FUNCTION_BLOCK "FB_Map_Siwarex_Core"
TITLE = Маппинг данных Siwarex CS
{ S7_Optimized_Access := 'FALSE' }
AUTHOR : S7C_Lib
FAMILY : Analog
VERSION : 1.4
// ==============================================================================
// Описание: Адаптированный маппинг из UDT_SIWA_CS. Обработка раздельных кодов
//           ошибок (модуля и драйвера). Встроенный таймер Watchdog в STAT.
// ==============================================================================
   VAR
      stat_Diag_CS_1 { ExternalAccessible := 'False'; ExternalVisible := 'False'; ExternalWritable := 'False'} : Struct   // Внутренняя память для Watchdog
         Old_Count { ExternalAccessible := 'False'; ExternalVisible := 'False'; ExternalWritable := 'False'} : Byte;
         Old_Weight { ExternalAccessible := 'False'; ExternalVisible := 'False'; ExternalWritable := 'False'} : Real;
         Last_Change_ms { ExternalAccessible := 'False'; ExternalVisible := 'False'; ExternalWritable := 'False'} : Real;
      END_STRUCT;
      stat_Diag_CS_2 { ExternalAccessible := 'False'; ExternalVisible := 'False'; ExternalWritable := 'False'} : Struct   // Внутренняя память для Watchdog
         Old_Count { ExternalAccessible := 'False'; ExternalVisible := 'False'; ExternalWritable := 'False'} : Byte;
         Old_Weight { ExternalAccessible := 'False'; ExternalVisible := 'False'; ExternalWritable := 'False'} : Real;
         Last_Change_ms { ExternalAccessible := 'False'; ExternalVisible := 'False'; ExternalWritable := 'False'} : Real;
      END_STRUCT;
   END_VAR

   VAR_TEMP
      temp_Value_Changed : Bool;
      temp_Counter_Changed : Bool;
   END_VAR


BEGIN

	// ============================================================================
	// SCALE CS_1
	// ============================================================================

	// 1. Веса
	"DB_MAP".Scale_CS_1.Weight_Gross_kg := INT_TO_REAL("DB_SCALE_CS_1".s_PROCESS_VALUES.i_GROSS_WEIGHT_PROC);
	"DB_MAP".Scale_CS_1.Weight_Net_kg := INT_TO_REAL("DB_SCALE_CS_1".s_PROCESS_VALUES.i_NET_WEIGHT_PROC);
	"DB_MAP".Scale_CS_1.Weight_Tare_kg := INT_TO_REAL("DB_SCALE_CS_1".s_PROCESS_VALUES.i_TARE_WEIGHT_PROC);

	// 2. Статусы
	"DB_MAP".Scale_CS_1.Status.Standstill := "DB_SCALE_CS_1".s_PROCESS_VALUES.bo_STA_ST_STAND_SCALE_ON;
	"DB_MAP".Scale_CS_1.Status.Limit_1 := "DB_SCALE_CS_1".s_PROCESS_VALUES.bo_STA_LIMIT1_ON;
	"DB_MAP".Scale_CS_1.Status.Limit_2 := "DB_SCALE_CS_1".s_PROCESS_VALUES.bo_STA_LIMIT2_ON;
	"DB_MAP".Scale_CS_1.Status.Tared := "DB_SCALE_CS_1".s_PROCESS_VALUES.bo_STA_TARED;
	"DB_MAP".Scale_CS_1.Status.Quarter_D_Zero := "DB_SCALE_CS_1".s_PROCESS_VALUES.bo_STA_025_D_ZERO;
	"DB_MAP".Scale_CS_1.Status.Scale_Calibrated := "DB_SCALE_CS_1".s_PROCESS_VALUES.bo_STA_SCALE_CALIBRATED;
	"DB_MAP".Scale_CS_1.Status.Write_Protected := "DB_SCALE_CS_1".s_PROCESS_VALUES.bo_STA_WRI_PROT;
	"DB_MAP".Scale_CS_1.Status.Limit_Max := "DB_SCALE_CS_1".s_PROCESS_VALUES.bo_STA_MAX_9E;
	"DB_MAP".Scale_CS_1.Status.Fault_HW := "DB_SCALE_CS_1".s_PROCESS_VALUES.bo_STA_ERROR_ON;
	"DB_MAP".Scale_CS_1.Status.Fault_FB := "DB_SCALE_CS_1".bo_FB_ERR;
	"DB_MAP".Scale_CS_1.Status.Fault := "DB_SCALE_CS_1".s_PROCESS_VALUES.bo_STA_ERROR_ON OR "DB_SCALE_CS_1".bo_FB_ERR;

	// 3. Коды ошибок: старший байт = b_OPR_ERR_MSG, младший = b_FB_ERR_CODE
	"DB_MAP".Scale_CS_1.Err_Raw :=
	    SHL(IN := BYTE_TO_WORD("DB_SCALE_CS_1".s_PROCESS_VALUES.b_OPR_ERR_MSG), N := 8)
	    OR BYTE_TO_WORD("DB_SCALE_CS_1".b_FB_ERR_CODE);

	// 4. Watchdog CS_1
	#temp_Value_Changed := ("DB_MAP".Scale_CS_1.Weight_Net_kg <> #stat_Diag_CS_1.Old_Weight);
	#temp_Counter_Changed := ("DB_SCALE_CS_1".b_INFO_REFRESH_COUNT <> #stat_Diag_CS_1.Old_Count);

	IF #temp_Counter_Changed THEN //#temp_Value_Changed OR
	    #stat_Diag_CS_1.Last_Change_ms := 0.0;
	    #stat_Diag_CS_1.Old_Weight := "DB_MAP".Scale_CS_1.Weight_Net_kg;
	    #stat_Diag_CS_1.Old_Count := "DB_SCALE_CS_1".b_INFO_REFRESH_COUNT;
	    "DB_MAP".Scale_CS_1.Status.Comm_Fault := FALSE;
	ELSE
	    #stat_Diag_CS_1.Last_Change_ms := #stat_Diag_CS_1.Last_Change_ms + "getCycleTime"();
	    IF #stat_Diag_CS_1.Last_Change_ms > 5000.0 THEN
	        "DB_MAP".Scale_CS_1.Status.Comm_Fault := TRUE;
	    END_IF;
	END_IF;


	// ============================================================================
	// SCALE CS_2
	// ============================================================================

	// 1. Веса
	"DB_MAP".Scale_CS_2.Weight_Gross_kg := INT_TO_REAL("DB_SCALE_CS_2".s_PROCESS_VALUES.i_GROSS_WEIGHT_PROC);
	"DB_MAP".Scale_CS_2.Weight_Net_kg := INT_TO_REAL("DB_SCALE_CS_2".s_PROCESS_VALUES.i_NET_WEIGHT_PROC);
	"DB_MAP".Scale_CS_2.Weight_Tare_kg := INT_TO_REAL("DB_SCALE_CS_2".s_PROCESS_VALUES.i_TARE_WEIGHT_PROC);

	// 2. Статусы
	"DB_MAP".Scale_CS_2.Status.Standstill := "DB_SCALE_CS_2".s_PROCESS_VALUES.bo_STA_ST_STAND_SCALE_ON;
	"DB_MAP".Scale_CS_2.Status.Limit_1 := "DB_SCALE_CS_2".s_PROCESS_VALUES.bo_STA_LIMIT1_ON;
	"DB_MAP".Scale_CS_2.Status.Limit_2 := "DB_SCALE_CS_2".s_PROCESS_VALUES.bo_STA_LIMIT2_ON;
	"DB_MAP".Scale_CS_2.Status.Tared := "DB_SCALE_CS_2".s_PROCESS_VALUES.bo_STA_TARED;
	"DB_MAP".Scale_CS_2.Status.Quarter_D_Zero := "DB_SCALE_CS_2".s_PROCESS_VALUES.bo_STA_025_D_ZERO;
	"DB_MAP".Scale_CS_2.Status.Scale_Calibrated := "DB_SCALE_CS_2".s_PROCESS_VALUES.bo_STA_SCALE_CALIBRATED;
	"DB_MAP".Scale_CS_2.Status.Write_Protected := "DB_SCALE_CS_2".s_PROCESS_VALUES.bo_STA_WRI_PROT;
	"DB_MAP".Scale_CS_2.Status.Limit_Max := "DB_SCALE_CS_2".s_PROCESS_VALUES.bo_STA_MAX_9E;
	"DB_MAP".Scale_CS_2.Status.Fault_HW := "DB_SCALE_CS_2".s_PROCESS_VALUES.bo_STA_ERROR_ON;
	"DB_MAP".Scale_CS_2.Status.Fault_FB := "DB_SCALE_CS_2".bo_FB_ERR;
	"DB_MAP".Scale_CS_2.Status.Fault := "DB_SCALE_CS_2".s_PROCESS_VALUES.bo_STA_ERROR_ON OR "DB_SCALE_CS_2".bo_FB_ERR;
	// 3. Коды ошибок
	"DB_MAP".Scale_CS_2.Err_Raw :=
	SHL(IN := BYTE_TO_WORD("DB_SCALE_CS_2".s_PROCESS_VALUES.b_OPR_ERR_MSG), N := 8)
	OR BYTE_TO_WORD("DB_SCALE_CS_2".b_FB_ERR_CODE);

	// 4. Watchdog CS_2
	#temp_Value_Changed := ("DB_MAP".Scale_CS_2.Weight_Net_kg <> #stat_Diag_CS_2.Old_Weight);
	#temp_Counter_Changed := ("DB_SCALE_CS_2".b_INFO_REFRESH_COUNT <> #stat_Diag_CS_2.Old_Count);

	IF #temp_Counter_Changed THEN //#temp_Value_Changed OR
	    #stat_Diag_CS_2.Last_Change_ms := 0.0;
	    #stat_Diag_CS_2.Old_Weight := "DB_MAP".Scale_CS_2.Weight_Net_kg;
	    #stat_Diag_CS_2.Old_Count := "DB_SCALE_CS_2".b_INFO_REFRESH_COUNT;
	    "DB_MAP".Scale_CS_2.Status.Comm_Fault := FALSE;
	ELSE
	    #stat_Diag_CS_2.Last_Change_ms := #stat_Diag_CS_2.Last_Change_ms + "getCycleTime"();
	    IF #stat_Diag_CS_2.Last_Change_ms > 5000.0 THEN
	        "DB_MAP".Scale_CS_2.Status.Comm_Fault := TRUE;
	    END_IF;
	END_IF;

END_FUNCTION_BLOCK

